{attribute 'qualified_only' := ''}
{attribute 'strict' := ''}
TYPE MC_StartMode :
(
	mcAbsolute := 0,
	mcRelative := 1,
	mcRampIn := 2
);
END_TYPE

(* stored: Version 1.1.0.1, ProductVersion 3.1.4024.12
   DUT MC_StartMode: Id {ed149f0d-703b-4c9e-a97b-29c6ab639eb6} *)
